Fanuc KAREL source: kt00517.KL

-- PROVISIONAL review KL for V1013-1; original PC SHA256 8d52a5c8ea74a26bf5c8c42162451e9ad66e1f3f2032fa86ceb471fc20b9b21a
-- Incomplete behavior may be omitted. Consult companion uncertainty JSON. Do not deploy.
PROGRAM KT00517
%NOLOCKGROUP
-- UNRESOLVED_DECL P1 type=000106
-- UNRESOLVED_DECL P2 type=000101
-- UNRESOLVED_DECL OUT type=000199
BEGIN
  -- UNRESOLVED_PC offsets 5-20; opcodes 2E,22,32,35
  -- UNRESOLVED_PC offsets 25-59; opcodes 49,7E,49,60,7E,4A
  -- UNRESOLVED_PC offsets 64-68; opcodes 7F
END KT00517
